(* CoDeSys 2.3 export: FK15PUMPSFAULTYCONTROL.EXP *)

(* POU K15/fK15PumpsFaultyControl, ST *)
FUNCTION fK15PumpsFaultyControl :BOOL
(* Проверка состояния насосов*)
VAR_INPUT
	PumpState : ARRAY [1..MAX_K15_PUMPS_NUM] OF BOOL;
	PumpStatusCheckDelay : ARRAY [1..MAX_K15_PUMPS_NUM] OF BOOL;
	PressureDrop : BOOL;
	EmergencyPumpStopButtonPressed: ARRAY [1..MAX_K15_PUMPS_NUM] OF BOOL; (*Нажат аварийный стоп насоса?*)
END_VAR
VAR
	i : USINT;
	activePumpID : USINT; (*номер работающего насоса*)
END_VAR
activePumpID := 0;

FOR i := 1 TO MAX_K15_PUMPS_NUM DO
	IF PumpState[i] THEN
		IF activePumpID > 1 THEN
			(*
				Включено больше одного насоса -
				ничего не можем сказать об их исправности
			*)
			RETURN;
		END_IF;
		activePumpID := activePumpID + 1;
	END_IF;
END_FOR;

IF activePumpID = 0 THEN
	(*
		Не включен ни один насос - 
		ничего не можем сказать об их исправности
	*)
	RETURN;
END_IF;

IF PumpStatusCheckDelay[activePumpID] THEN
	(*
		Определяем исправность насоса
		по перепаду давления
	*)
	K15PumpFaulty[activePumpID] := NOT(PressureDrop);
	IF EmergencyPumpStopButtonPressed[activePumpID] THEN
 		K15PumpFaulty[activePumpID] := TRUE;
	END_IF;
END_IF;
END_FUNCTION
